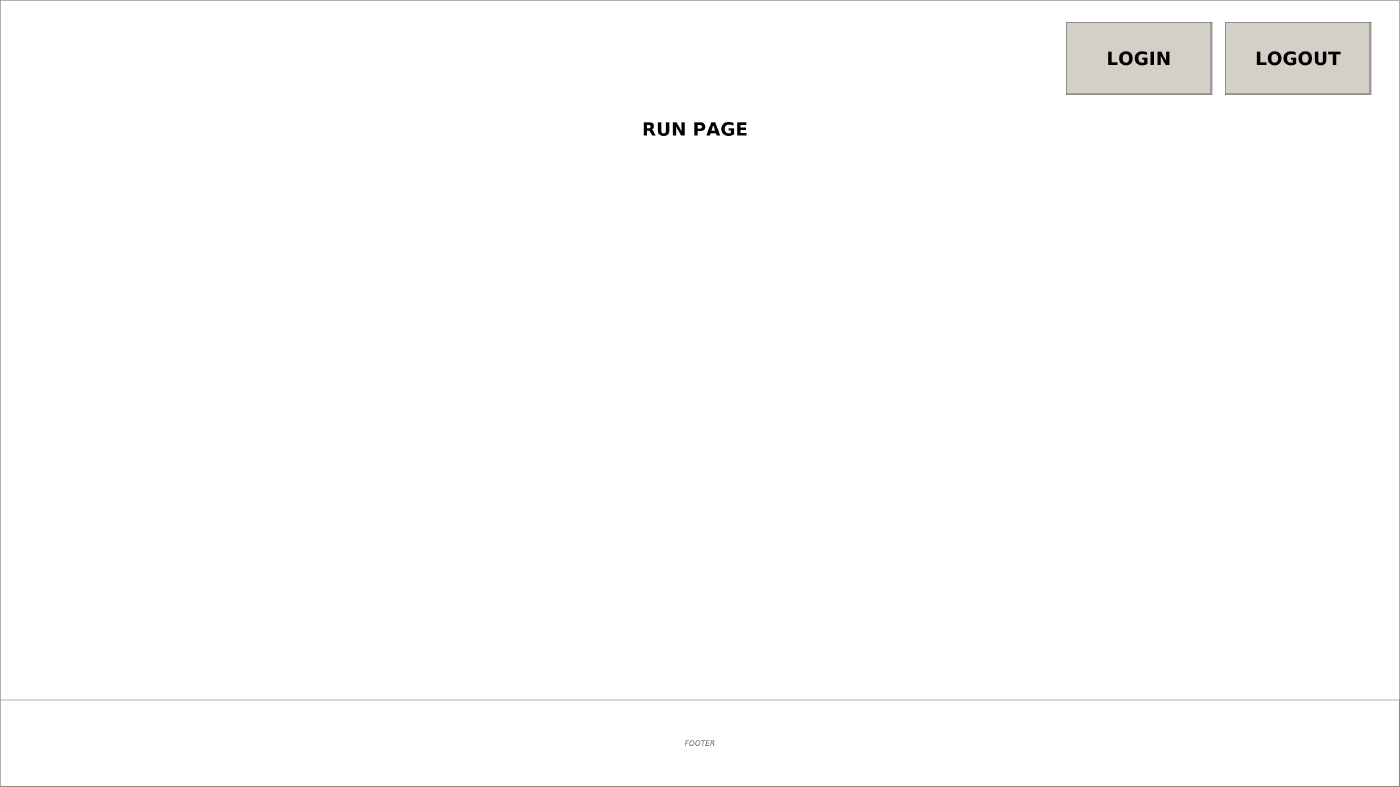
VISUALIZATION PAGE_RUN  // 1920x1080, background image ImagePool.Grey_Gradient
    Button (1462,30 200x100), "LOGIN"
        OnMouseClick: VisuUserMgmt Type=Login
    Button (1680,30 200x100), "LOGOUT"
        OnMouseClick: VisuUserMgmt Type=Logout
    Frame (0,960 1920x120)
        shows FOOTER()
    Label (718,119 470x116), "RUN PAGE"
END_VISUALIZATION

(* stored: Version 1.1.0.1, ProductVersion 3.1.4024.12
   Visu PAGE_RUN: Id {21aefe76-6c90-4971-be64-d5e2d4a32b67} *)
